// TwinCAT 3 PLC project RoomController
// ProgramVersion: 3.1.4023.0
// libraries:
//   Tc2_Standard, * (Beckhoff Automation GmbH)
//   Tc2_System, * (Beckhoff Automation GmbH)
//   Tc3_Module, * (Beckhoff Automation GmbH)
// project tree:
//   DUTs/ stAi8CH.TcDUT, stRoomData.TcDUT
//   GVLs/ IO.TcGVL
//   / PlcTask.TcTTO (not stored)
//   POUs/ fbIntValueSimulation.TcPOU, Hardware_Simulation.TcPOU, MAIN.TcPOU
// real-time tasks:
//   TASK PlcTask: cycle T#10ms, priority 20, ADS port 350
// I/O:
//   DEVICE Device 1 (EtherCAT) (disabled), AmsNetId 172.20.10.241.2.1
//     Term 1 (EK1200) [EK1200-5000 EtherCAT Power supply (2A E-Bus)]
//       Term 2 (EL3164) [EL3164 4Ch. Ana. Input 0-10V]
//       Term 3 (EL9011) [EL9011 End Terminal]
// variable links:
//   RoomController/RoomController Instance <-> Device 1 (EtherCAT)/Term 1 (EK1200)/Term 2 (EL3164)
//     PlcTask Inputs/IO.hwAirDataIN.CH{1..4} <-> AI Standard Channel {1..4}/Value  (4 links)

// ---- DUTs/stAi8CH.TcDUT
TYPE stAi8CH :
STRUCT
	CH1 AT %I* : INT;
	CH2 AT %I* : INT;
	CH3 AT %I* : INT;
	CH4 AT %I* : INT;
	CH5 AT %I* : INT;
	CH6 AT %I* : INT;
	CH7 AT %I* : INT;
	CH8 AT %I* : INT;
	
END_STRUCT
END_TYPE

// ---- DUTs/stRoomData.TcDUT
TYPE stRoomData :
STRUCT
	{attribute addProperty Name "<#Actual room temperature °C#>"}
	Temperature : REAL;
	{attribute addProperty Name "<#Actual room humidity %#>"}
	Humidity : REAL;
	{attribute addProperty Name "<#Actual room VOC %#>"}
	VOC : REAL;
	{attribute addProperty Name "<#Actual room CO2 concentration ppm#>"}
	CO2 : REAL;
	{attribute addProperty Name "<#Actual room absolute humidity g/m3#>"}
	AbsoluteHumidity : REAL;
	{attribute addProperty Name "<#Actual room enthalpy kJ/k#>"}
	Enthalpy : REAL;
	{attribute addProperty Name "<#Actual room dew point °C#>"}
	DewPoint : REAL;
	{attribute addProperty Name "<#Actual room CO2 VOC mix#>"}
	CO2VOC_MIX : REAL;
END_STRUCT
END_TYPE

// ---- GVLs/IO.TcGVL
{attribute 'qualified_only'}
VAR_GLOBAL
	hwAirDataIN : stAi8CH;
END_VAR

// ---- POUs/fbIntValueSimulation.TcPOU
FUNCTION_BLOCK fbIntValueSimulation
VAR_INPUT
	MinValue : INT;
	MaxValue : INT;
END_VAR
VAR_IN_OUT
	Value : INT;
END_VAR
VAR
	p1 : INT :=2;
	p2 : INT :=1;
	pm : INT;
	x0 : INT;
END_VAR

x0 := Value;
pm := MaxValue-MinValue;
IF x0 = 0 THEN
	x0 := (MaxValue + MinValue) / 2;
END_IF

Value := MinValue + ((x0*p1 + p2) MOD pm);

END_FUNCTION_BLOCK

// ---- POUs/Hardware_Simulation.TcPOU
PROGRAM Hardware_Simulation
VAR
	CH1 : fbIntValueSimulation;
	CH2 : fbIntValueSimulation;
	CH3 : fbIntValueSimulation;
	CH4 : fbIntValueSimulation;
	
	CH5 : fbIntValueSimulation;
	CH6 : fbIntValueSimulation;
	CH7 : fbIntValueSimulation;
	CH8 : fbIntValueSimulation;
END_VAR

CH1(MinValue := 16000 , MaxValue := 16500 , Value := IO.hwAirDataIN.CH1);
CH2(MinValue := 9800 , MaxValue := 10000 , Value := IO.hwAirDataIN.CH2);
CH3(MinValue := 300 , MaxValue := 350 , Value := IO.hwAirDataIN.CH3);
CH4(MinValue := 3600 , MaxValue := 3700 , Value := IO.hwAirDataIN.CH4);

CH5(MinValue := 2620 , MaxValue := 2650 , Value := IO.hwAirDataIN.CH5);
CH6(MinValue := 10000 , MaxValue := 10500 , Value := IO.hwAirDataIN.CH6);
CH7(MinValue := 3930 , MaxValue := 4000 , Value := IO.hwAirDataIN.CH7);
CH8(MinValue := 6000 , MaxValue := 6200 , Value := IO.hwAirDataIN.CH8);

END_PROGRAM

// ---- POUs/MAIN.TcPOU
PROGRAM MAIN
VAR
	RoomData : stRoomData;
END_VAR

Hardware_Simulation();

RoomData.Temperature := INT_TO_REAL(IO.hwAirDataIN.CH1) / 32767 * 50.0; // as 0-10V~0-32767~0-50°C
RoomData.Humidity := INT_TO_REAL(IO.hwAirDataIN.CH2) / 32767 * 100.0; // as 0-10V~0-32767~0-100%
RoomData.VOC := INT_TO_REAL(IO.hwAirDataIN.CH3) / 32767 * 100.0; // as 0-10V~0-32767~0-100%
RoomData.CO2 := INT_TO_REAL(IO.hwAirDataIN.CH4) / 32767 * 5000.0; // as 0-10V~0-32767~0-5000ppm

RoomData.AbsoluteHumidity := INT_TO_REAL(IO.hwAirDataIN.CH5) / 32767 * 10.0; // as 0-10V~0-32767~0-10 g/m3
RoomData.Enthalpy := INT_TO_REAL(IO.hwAirDataIN.CH6) / 32767 * 100.0; // as 0-10V~0-32767~0-100 kJ/kg
RoomData.DewPoint := INT_TO_REAL(IO.hwAirDataIN.CH7) / 32767 * 50.0; // as 0-10V~0-32767~0-50 °C
RoomData.CO2VOC_MIX := INT_TO_REAL(IO.hwAirDataIN.CH8) / 32767 * 50.0; // as 0-10V~0-32767~0-50

END_PROGRAM
